{attribute 'qualified_only'}
VAR_GLOBAL PERSISTENT RETAIN
	
    stStatistics 				: ST_HmiStatistics;
    astEventsHistory 			: ARRAY[0..200] OF ST_EventsHistory;
	astTestHistory 				: ARRAY[0..2000] OF ST_TestHistory;
	uiTestHistoryWriteIndex 	: UINT := 0;
	uiTestHistoryCount      	: UINT := 0;
	
	stSiliconeSupply : ST_SiliconeSupplyPersistent := (
		aReservoirDegassed := [FALSE, FALSE],
		usiSelectedReservoir := 1
	);
	
END_VAR

(* stored: Version 1.1.0.1, ProductVersion 3.1.4026.18
   GVL GVL_Persistent: Id {3f671271-ab6d-41c2-a99c-4446f117874d} *)
